{attribute 'GeneratedUsingTerminal: EK1122-0000-0018'}
{attribute addProperty BoxType "EK1122-0000-0018"}
{attribute addProperty Id "Beckhoff_EL3xxx_0030sub_EK1100EK1100_1FC0878B2"}
{attribute addProperty CRC "1440408522"}
{attribute addProperty Size "2"}
TYPE Beckhoff_EL3xxx_0030EK1122_55DAE3CA EXTENDS EK1122_1FC0878B :
STRUCT
	{attribute addProperty Name "Beckhoff_EL3xxx_0030sub_EK1100"}
	{attribute addProperty PreviousPort "Beckhoff EL3xxx-0030EK1122 : D"}
	Beckhoff_EL3xxx_0030sub_EK1100 : EK1100_1FC0878B;
END_STRUCT
END_TYPE

(* stored: Version 1.2.0.0, ProductVersion 3.1.4024.9
   DUT Beckhoff_EL3xxx_0030EK1122_55DAE3CA: Id {dfd0fa87-942d-4a6a-a432-55edc338c13c} *)
